// TIA Portal project "FactoryIO_Template_S7-1500_V15_V15.1" (V15.1)

(* hardware
DEVICE "S71500/ET200MP-Station_1"  S7-1500 station
   slot 0: "Profilschiene_0"  6ES7 590-1***0-0AA0
   slot 1: "PLC_1"  CPU 1511-1 PN  6ES7 511-1AK00-0AB0  V1.8
   slot 2: "AI 8xU/I/RTD/TC ST_1"  AI 8xU/I/RTD/TC ST  6ES7 531-7KF00-0AB0  V2.0
   slot 3: "AI 8xU/I/RTD/TC ST_2"  AI 8xU/I/RTD/TC ST  6ES7 531-7KF00-0AB0  V2.0
   slot 4: "AI 8xU/I/RTD/TC ST_3"  AI 8xU/I/RTD/TC ST  6ES7 531-7KF00-0AB0  V2.0
   slot 5: "AI 8xU/I/RTD/TC ST_4"  AI 8xU/I/RTD/TC ST  6ES7 531-7KF00-0AB0  V2.0
   slot 6: "DI 16x24VDC BA_1"  DI 16x24VDC BA  6ES7 521-1BH10-0AA0  V1.0
*)

// ===== PLC "PLC_1"  CPU 1511-1 PN =====

VAR_GLOBAL   // PLC tag table "Standard-Variablentabelle"
   "HighSensor" AT %E0.0 : Bool;
   "LowSensor" AT %I0.1 : Bool;
   "PalletSensor" AT %I0.2 : Bool;
   "Loaded" AT %I0.3 : Bool;
   "AtLeftEntry" AT %I0.4 : Bool;
   "AtLeftExit" AT %I0.5 : Bool;
   "AtRightEntry" AT %I0.6 : Bool;
   "AtRightExit" AT %I0.7 : Bool;
   "Start" AT %I1.0 : Bool;
   "Reset" AT %I1.1 : Bool;
   "Stop" AT %I1.2 : Bool;
   "EmergencyStop" AT %I1.3 : Bool;
   "Auto" AT %I1.4 : Bool;
   "Load" AT %Q0.1 : Bool;
   "Unload" AT %Q0.2 : Bool;
   "Transf. Left" AT %Q0.3 : Bool;
   "Transf. Right" AT %Q0.4 : Bool;
   "Conveyor Left" AT %Q0.5 : Bool;
   "Conveyor Right" AT %Q0.6 : Bool;
   "Start Light" AT %Q0.7 : Bool;
   "Reset Light" AT %Q1.0 : Bool;
   "Stop Light" AT %Q1.1 : Bool;
   "Counter" AT %QW30 : Int;
   "Conveyor Entry" AT %Q0.0 : Bool;
   "DelayReset" AT %T0 : Timer;
   "DelayTransferencia" AT %T1 : Timer;
END_VAR

TYPE "ControleDeCiclo"
   STRUCT
      Ciclo_Inicado : Bool;
      Em_Parada : Bool;
      Reset : Bool;
      Em_Manual : Bool;
      Em_Automatico : Bool;
      Counter_Entrada : Bool;
      Em_Anomali : Bool;
   END_STRUCT;
END_TYPE

// folder: SortByHeight

DATA_BLOCK "Painel_DB"   // DB1
{ S7_Optimized_Access := 'TRUE' }
VERSION : 0.1
// stored: InstanceOfName Painel
"Painel"
BEGIN
END_DATA_BLOCK

DATA_BLOCK "Conveyor_Entry_DB"   // DB2
{ S7_Optimized_Access := 'TRUE' }
VERSION : 0.1
// stored: InstanceOfName Conveyor_Entry
"Conveyor_Entry"
BEGIN
END_DATA_BLOCK

DATA_BLOCK "Controle_Sentido_DB"   // DB3
{ S7_Optimized_Access := 'TRUE' }
VERSION : 0.1
// stored: InstanceOfName Controle_Sentido
"Controle_Sentido"
BEGIN
END_DATA_BLOCK

// folder: (top level)

FUNCTION "MHJ-PLC-Lab-Function-S71500" : Void   // FC9000, SCL
{ S7_Optimized_Access := 'TRUE' }
VERSION : 0.1
   VAR_TEMP
      Value : Byte;
      ForCounter : Int;
   END_VAR
   VAR CONSTANT
      Value_01_DW : DWord := 16#1223_5486;
      Value_02_DW : DWord := 16#A6C9_D1F5;
   END_VAR
BEGIN

   #Value:=PEEK(area := 16#82,
        dbNumber := 0,
        byteOffset := 511);
   #Value := #Value + 1;

   POKE(area := 16#82,
        dbNumber := 0,
        byteOffset := 511,
        value := #Value);

   POKE(area := 16#82,
        dbNumber := 0,
        byteOffset := 1016,
        value := #Value_01_DW);
   POKE(area := 16#82,
        dbNumber := 0,
        byteOffset := 1020,
        value := #Value_02_DW);

   FOR #ForCounter := 0 TO 63 DO
       #Value:=PEEK(area := 16#1,
            dbNumber := 0,
            byteOffset := #ForCounter);
       POKE(area := 16#81,
            dbNumber := 0,
            byteOffset := #ForCounter,
            value := #Value);
   END_FOR;
   #Value := PEEK(area := 16#1,
                  dbNumber := 0,
                  byteOffset := 512);
   POKE(area := 16#82,
        dbNumber := 0,
        byteOffset := 512,
        value := #Value);
END_FUNCTION

ORGANIZATION_BLOCK "Main"   // OB1, FBD, ProgramCycle
TITLE = "Main Program Sweep (Cycle)"
{ S7_Optimized_Access := 'TRUE' }
VERSION : 0.1
   VAR_INPUT
      Initial_Call : Bool;   // Initial call of this OB
      Remanence : Bool;   // =True, if remanent data are available
   END_VAR
BEGIN

REGION Network 1
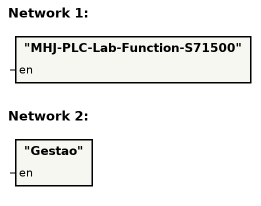
   "MHJ-PLC-Lab-Function-S71500"();
END_REGION

REGION Network 2
   "Gestao"();
END_REGION
END_ORGANIZATION_BLOCK

// folder: SortByHeight

FUNCTION "Gestao" : Void   // FC1, LAD
{ S7_Optimized_Access := 'TRUE' }
VERSION : 0.1
BEGIN

REGION Network 1
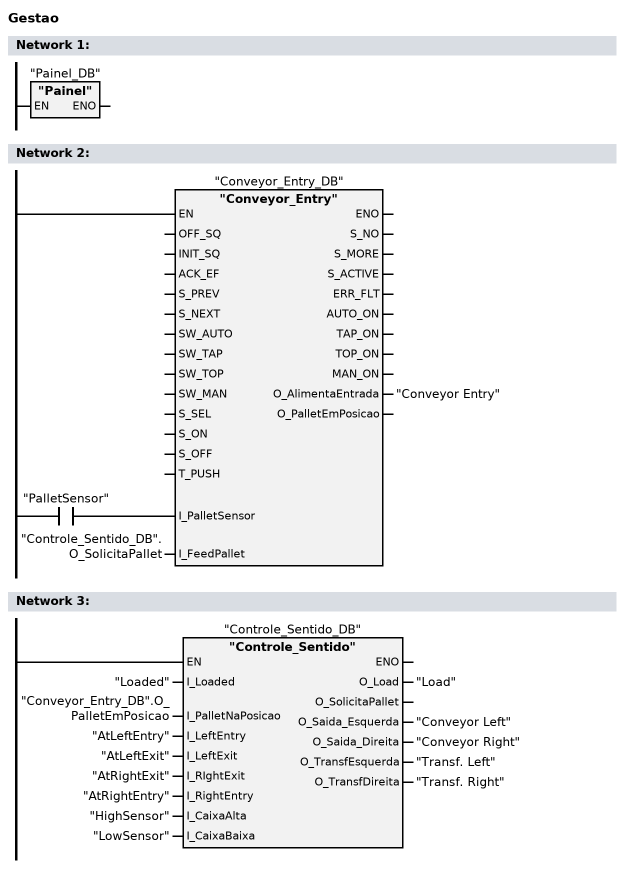
   RUNG wire#powerrail
      "Painel_DB"()
   END_RUNG
   // the same network as SCL:
   "Painel_DB"();   // "Painel"
END_REGION

REGION Network 2
   RUNG wire#powerrail
      "Conveyor_Entry_DB"(I_PalletSensor := wire#w1, OFF_SQ :=, INIT_SQ :=, ACK_EF :=, S_PREV :=, S_NEXT :=, SW_AUTO :=, SW_TAP :=, SW_TOP :=, SW_MAN :=, S_SEL :=, S_ON :=, S_OFF :=, T_PUSH :=, I_FeedPallet := "Controle_Sentido_DB".O_SolicitaPallet, S_NO =>, S_MORE =>, S_ACTIVE =>, ERR_FLT =>, AUTO_ON =>, TAP_ON =>, TOP_ON =>, MAN_ON =>, O_AlimentaEntrada => "Conveyor Entry", O_PalletEmPosicao =>)
   END_RUNG
   RUNG wire#powerrail
      Contact( "PalletSensor" )
   END_RUNG wire#w1
   // the same network as SCL:
   "Conveyor_Entry_DB"(I_PalletSensor := "PalletSensor",   // "Conveyor_Entry"
                       I_FeedPallet := "Controle_Sentido_DB".O_SolicitaPallet,
                       O_AlimentaEntrada => "Conveyor Entry");
END_REGION

REGION Network 3
   RUNG wire#powerrail
      "Controle_Sentido_DB"(I_Loaded := "Loaded", I_PalletNaPosicao := "Conveyor_Entry_DB".O_PalletEmPosicao, I_LeftEntry := "AtLeftEntry", I_LeftExit := "AtLeftExit", I_RIghtExit := "AtRightExit", I_RightEntry := "AtRightEntry", I_CaixaAlta := "HighSensor", I_CaixaBaixa := "LowSensor", O_Load => "Load", O_SolicitaPallet =>, O_Saida_Esquerda => "Conveyor Left", O_Saida_Direita => "Conveyor Right", O_TransfEsquerda => "Transf. Left", O_TransfDireita => "Transf. Right")
   END_RUNG
   // the same network as SCL:
   "Controle_Sentido_DB"(I_Loaded := "Loaded",   // "Controle_Sentido"
                         I_PalletNaPosicao := "Conveyor_Entry_DB".O_PalletEmPosicao,
                         I_LeftEntry := "AtLeftEntry",
                         I_LeftExit := "AtLeftExit",
                         I_RIghtExit := "AtRightExit",
                         I_RightEntry := "AtRightEntry",
                         I_CaixaAlta := "HighSensor",
                         I_CaixaBaixa := "LowSensor",
                         O_Load => "Load",
                         O_Saida_Esquerda => "Conveyor Left",
                         O_Saida_Direita => "Conveyor Right",
                         O_TransfEsquerda => "Transf. Left",
                         O_TransfDireita => "Transf. Right");
END_REGION
END_FUNCTION

// folder: SortByHeight/ControleSentido

FUNCTION_BLOCK "Controle_Sentido"   // FB3, LAD
{ S7_Optimized_Access := 'TRUE' }
VERSION : 0.1
   VAR_INPUT
      I_Loaded : Bool;
      I_PalletNaPosicao : Bool;
      I_LeftEntry : Bool;
      I_LeftExit : Bool;
      I_RIghtExit : Bool;
      I_RightEntry : Bool;
      I_CaixaAlta : Bool;
      I_CaixaBaixa : Bool;
   END_VAR
   VAR_OUTPUT
      O_Load : Bool;
      O_SolicitaPallet : Bool;
      O_Saida_Esquerda : Bool;
      O_Saida_Direita : Bool;
      O_TransfEsquerda : Bool;
      O_TransfDireita : Bool;
   END_VAR
   VAR
      Abastecido : Bool;
      Desabastecido : Bool;
      Estado_Saida_Esquerda : Bool;
      Estado_Saida_Direita : Bool;
      "Caixa alta" : Bool;
      "Caixa baixa" : Bool;
      M1 : Bool;
      M2 : Bool;
      M3 : Bool;
      M4 : Bool;
      M5 : Bool;
      M6 : Bool;
      Transf_Esquerda : Bool;
      Transf_Direita : Bool;
      Em_Transferencia : Bool;
      StoptEsquerda : Bool;
      StoptDireita : Bool;
   END_VAR
   VAR_TEMP   // added for the SCL form of the ladder/FBD networks
      _w1 : Bool;
   END_VAR
BEGIN

REGION Network 1: ############## ABASTECIMENTO ################
END_REGION

REGION Network 2: Desabastecido
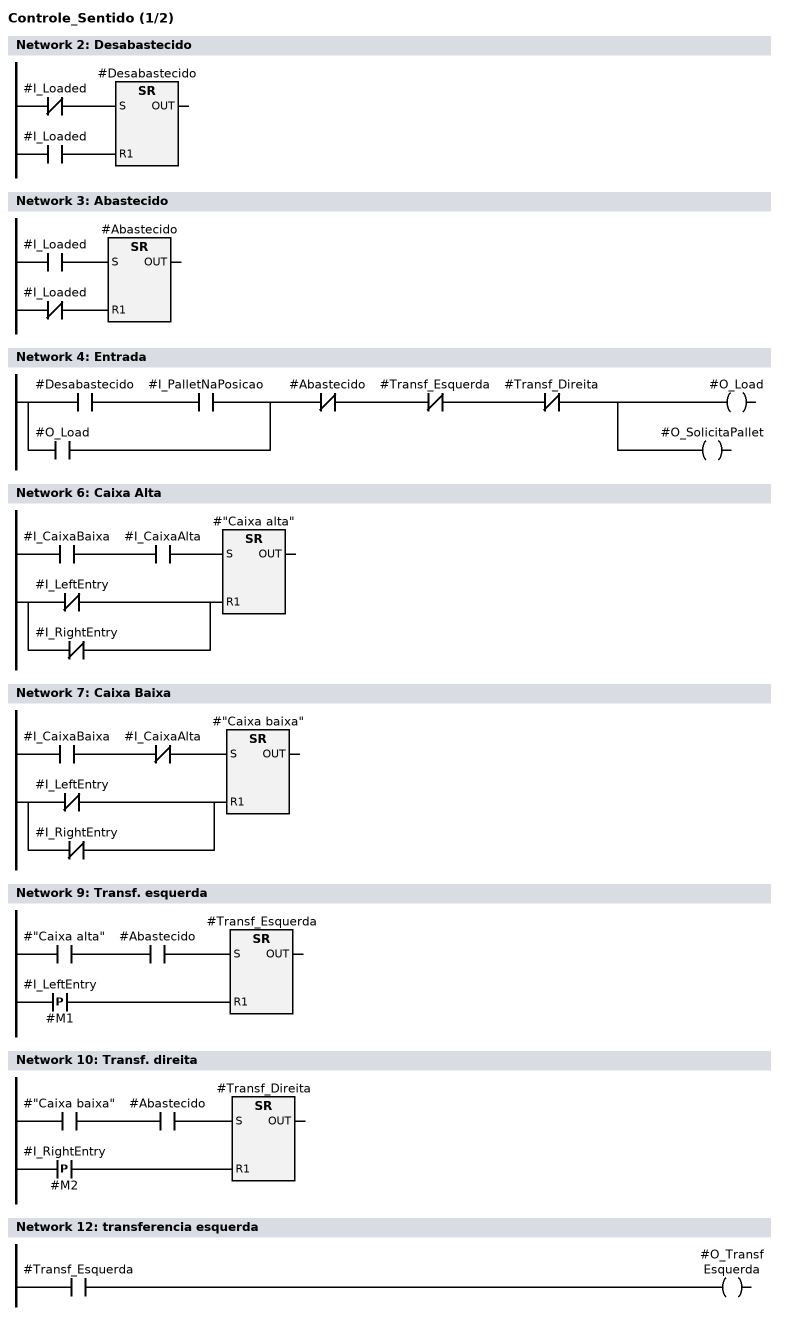
   RUNG wire#powerrail
      I_Contact( #I_Loaded )
      S_SR(operand := #Desabastecido, r1 := wire#w1)
   END_RUNG
   RUNG wire#powerrail
      Contact( #I_Loaded )
   END_RUNG wire#w1
   // the same network as SCL:
   IF NOT #I_Loaded THEN
       #Desabastecido := TRUE;   // SR flip-flop
   END_IF;
   IF #I_Loaded THEN #Desabastecido := FALSE; END_IF;
END_REGION

REGION Network 3: Abastecido
   RUNG wire#powerrail
      Contact( #I_Loaded )
      S_SR(operand := #Abastecido, r1 := wire#w1)
   END_RUNG
   RUNG wire#powerrail
      I_Contact( #I_Loaded )
   END_RUNG wire#w1
   // the same network as SCL:
   IF #I_Loaded THEN
       #Abastecido := TRUE;   // SR flip-flop
   END_IF;
   IF NOT #I_Loaded THEN #Abastecido := FALSE; END_IF;
END_REGION

REGION Network 4: Entrada
   RUNG wire#powerrail
      Contact( #Desabastecido )
      Contact( #I_PalletNaPosicao )
      wire#w1
      I_Contact( #Abastecido )
      I_Contact( #Transf_Esquerda )
      I_Contact( #Transf_Direita )
      wire#w2
      Coil( #O_Load )
   END_RUNG
   RUNG wire#powerrail
      Contact( #O_Load )
   END_RUNG wire#w1
   RUNG wire#w2
      Coil( #O_SolicitaPallet )
   END_RUNG
   // the same network as SCL:
   #O_Load := ((#Desabastecido AND #I_PalletNaPosicao) OR #O_Load) AND NOT #Abastecido AND NOT #Transf_Esquerda AND NOT #Transf_Direita;
   #O_SolicitaPallet := #O_Load;
END_REGION

REGION Network 5: ################ TAMANHOS #################
END_REGION

REGION Network 6: Caixa Alta
   RUNG wire#powerrail
      Contact( #I_CaixaBaixa )
      Contact( #I_CaixaAlta )
      S_SR(operand := #"Caixa alta", r1 := wire#w1)
   END_RUNG
   RUNG wire#powerrail
      I_Contact( #I_LeftEntry )
   END_RUNG wire#w1
   RUNG wire#powerrail
      I_Contact( #I_RightEntry )
   END_RUNG wire#w1
   // the same network as SCL:
   IF #I_CaixaBaixa AND #I_CaixaAlta THEN
       #"Caixa alta" := TRUE;   // SR flip-flop
   END_IF;
   IF NOT #I_LeftEntry OR NOT #I_RightEntry THEN #"Caixa alta" := FALSE; END_IF;
END_REGION

REGION Network 7: Caixa Baixa
   RUNG wire#powerrail
      Contact( #I_CaixaBaixa )
      I_Contact( #I_CaixaAlta )
      S_SR(operand := #"Caixa baixa", r1 := wire#w1)
   END_RUNG
   RUNG wire#powerrail
      I_Contact( #I_LeftEntry )
   END_RUNG wire#w1
   RUNG wire#powerrail
      I_Contact( #I_RightEntry )
   END_RUNG wire#w1
   // the same network as SCL:
   IF #I_CaixaBaixa AND NOT #I_CaixaAlta THEN
       #"Caixa baixa" := TRUE;   // SR flip-flop
   END_IF;
   IF NOT #I_LeftEntry OR NOT #I_RightEntry THEN #"Caixa baixa" := FALSE; END_IF;
END_REGION

REGION Network 8: ############## TRANFERENCIAS ################
END_REGION

REGION Network 9: Transf. esquerda
   RUNG wire#powerrail
      Contact( #"Caixa alta" )
      Contact( #Abastecido )
      S_SR(operand := #Transf_Esquerda, r1 := wire#w1)
   END_RUNG
   RUNG wire#powerrail
      P_Contact(operand := #I_LeftEntry, bit := #M1)
   END_RUNG wire#w1
   // the same network as SCL:
   #_w1 := #I_LeftEntry AND NOT #M1;   // rising edge of #I_LeftEntry
   #M1 := #I_LeftEntry;
   IF #"Caixa alta" AND #Abastecido THEN
       #Transf_Esquerda := TRUE;   // SR flip-flop
   END_IF;
   IF #_w1 THEN #Transf_Esquerda := FALSE; END_IF;
END_REGION

REGION Network 10: Transf. direita
   RUNG wire#powerrail
      Contact( #"Caixa baixa" )
      Contact( #Abastecido )
      S_SR(operand := #Transf_Direita, r1 := wire#w1)
   END_RUNG
   RUNG wire#powerrail
      P_Contact(operand := #I_RightEntry, bit := #M2)
   END_RUNG wire#w1
   // the same network as SCL:
   #_w1 := #I_RightEntry AND NOT #M2;   // rising edge of #I_RightEntry
   #M2 := #I_RightEntry;
   IF #"Caixa baixa" AND #Abastecido THEN
       #Transf_Direita := TRUE;   // SR flip-flop
   END_IF;
   IF #_w1 THEN #Transf_Direita := FALSE; END_IF;
END_REGION

REGION Network 11: ################# SAIDA ###################
END_REGION

REGION Network 12: transferencia esquerda
   RUNG wire#powerrail
      Contact( #Transf_Esquerda )
      Coil( #O_TransfEsquerda )
   END_RUNG
   // the same network as SCL:
   #O_TransfEsquerda := #Transf_Esquerda;
END_REGION

REGION Network 13: Conveyor esquerda
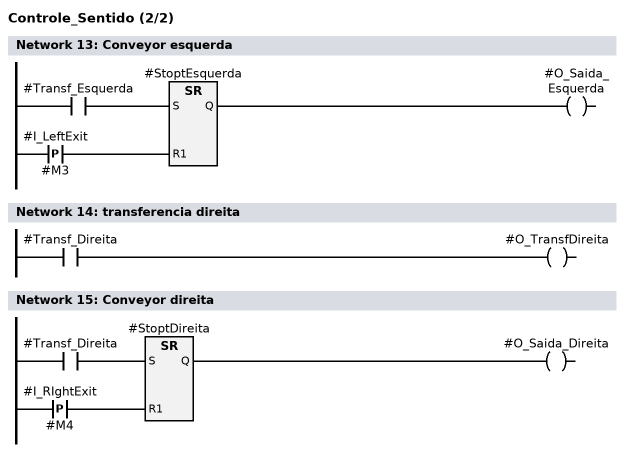
   RUNG wire#powerrail
      Contact( #Transf_Esquerda )
      S_SR(operand := #StoptEsquerda, r1 := wire#w1)
      Coil( #O_Saida_Esquerda )
   END_RUNG
   RUNG wire#powerrail
      P_Contact(operand := #I_LeftExit, bit := #M3)
   END_RUNG wire#w1
   // the same network as SCL:
   #_w1 := #I_LeftExit AND NOT #M3;   // rising edge of #I_LeftExit
   #M3 := #I_LeftExit;
   IF #Transf_Esquerda THEN
       #StoptEsquerda := TRUE;   // SR flip-flop
   END_IF;
   IF #_w1 THEN #StoptEsquerda := FALSE; END_IF;
   #O_Saida_Esquerda := #StoptEsquerda;
END_REGION

REGION Network 14: transferencia direita
   RUNG wire#powerrail
      Contact( #Transf_Direita )
      Coil( #O_TransfDireita )
   END_RUNG
   // the same network as SCL:
   #O_TransfDireita := #Transf_Direita;
END_REGION

REGION Network 15: Conveyor direita
   RUNG wire#powerrail
      Contact( #Transf_Direita )
      S_SR(operand := #StoptDireita, r1 := wire#w1)
      Coil( #O_Saida_Direita )
   END_RUNG
   RUNG wire#powerrail
      P_Contact(operand := #I_RIghtExit, bit := #M4)
   END_RUNG wire#w1
   // the same network as SCL:
   #_w1 := #I_RIghtExit AND NOT #M4;   // rising edge of #I_RIghtExit
   #M4 := #I_RIghtExit;
   IF #Transf_Direita THEN
       #StoptDireita := TRUE;   // SR flip-flop
   END_IF;
   IF #_w1 THEN #StoptDireita := FALSE; END_IF;
   #O_Saida_Direita := #StoptDireita;
END_REGION
END_FUNCTION_BLOCK

// folder: SortByHeight/ConveyorEntry

FUNCTION_BLOCK "Conveyor_Entry"   // FB2, GRAPH_PLUS
{ S7_Optimized_Access := 'TRUE' }
VERSION : 0.1
   VAR_INPUT
      OFF_SQ : Bool := false;   // Turn sequence off
      INIT_SQ : Bool := false;   // Set sequence to initial state
      ACK_EF : Bool := false;   // Acknowledge all errors and faults
      S_PREV : Bool := false;   // Output previous step in parameter S_NO
      S_NEXT : Bool := false;   // Indicate next step in parameter S_NO
      SW_AUTO : Bool := false;   // Automatic mode
      SW_TAP : Bool := false;   // Semiautomatic/switch with transition
      SW_TOP : Bool := false;   // Semiautomatic/ignore transition
      SW_MAN : Bool := false;   // Manual mode
      S_SEL : Int := 0;   // Select step to be output to S_NO
      S_ON : Bool := false;   // Activate step indicated in S_NO
      S_OFF : Bool := false;   // Deactivate step indicated S_NO
      T_PUSH : Bool := false;   // Enable transition to switch in semi automatic mode
      I_PalletSensor : Bool;
      I_FeedPallet : Bool;
   END_VAR
   VAR_OUTPUT
      S_NO : Int := 0;   // Step number
      S_MORE : Bool := false;   // More steps are available and can be shown in S_NO
      S_ACTIVE : Bool := false;   // Step indicated in S_NO is active
      ERR_FLT : Bool := false;   // Interlock or supervision group error
      AUTO_ON : Bool := false;   // Automatic mode is active
      TAP_ON : Bool := false;   // Semiautomatic mode/step with transition enabled
      TOP_ON : Bool := false;   // Semiautomatic mode/ignore transition enabled
      MAN_ON : Bool := false;   // Manual mode is active
      O_AlimentaEntrada : Bool;
      O_PalletEmPosicao : Bool;
   END_VAR
   VAR
      HMI_INFO : Array[0..8] of UInt;
      IF_PAR : G7_IfParPlus_V2;
      RT_DATA : G7_RTDataPlus_V2;   // Internal data area
      Trans4 : G7_TransitionPlus_V2;   // Transition structure
      Trans1 : G7_TransitionPlus_V2;   // Transition structure
      Trans2 : G7_TransitionPlus_V2;   // Transition structure
      Trans3 : G7_TransitionPlus_V2;   // Transition structure
      Step4 : G7_StepPlus_V2;   // Step structure
      Step1 : G7_StepPlus_V2;   // Step structure
      Step2 : G7_StepPlus_V2;   // Step structure
      Step3 : G7_StepPlus_V2;   // Step structure
      SINI : Array[0..1] of USInt;
      LSTT : Array[0..3] of USInt;
      ATAJ : Array[0..3] of USInt;
      ATAB : Array[0..3] of USInt;
      PSTT : Array[0..3] of USInt;
      NSTT : Array[0..3] of USInt;
      ASSJ : Array[0..3] of USInt;
      ASSB : Array[0..3] of USInt;
      PTTS : Array[0..3] of USInt;
      NTTS : Array[0..3] of USInt;
      SW_SQTS : Array[0..3] of USInt;
      SWITCH : Array[0..0] of USInt;
      TVX : Array[0..1] of USInt;
      TTX : Array[0..1] of USInt;
      TSX : Array[0..1] of USInt;
      S00X : Array[0..1] of USInt;
      SOFFX : Array[0..1] of USInt;
      SONX : Array[0..1] of USInt;
      SAX : Array[0..1] of USInt;
      SERRX : Array[0..4] of USInt;
      SMX : Array[0..4] of USInt;
      S0X : Array[0..4] of USInt;
      S1X : Array[0..4] of USInt;
      IL_ALARM_INST : Program_Alarm;
      SUP_ALARM_INST : Program_Alarm;
      STEP_TIME_ALARM_INST : Program_Alarm;
      IEC_TIMER_INST : IEC_TIMER;
      TRANSACTION_FLAG : Bool := false;
   END_VAR
   // LSTT[3] := 1;
   // SINI[0] := 2;
   // LSTT[0] := 255;
   // LSTT[1] := 255;
   // ATAJ[3] := 3;
   // ATAJ[1] := 1;
   // ATAJ[2] := 2;
   // ATAB[3] := 3;
   // ATAB[1] := 1;
   // ATAB[2] := 2;
   // PSTT[3] := 3;
   // PSTT[1] := 1;
   // PSTT[2] := 2;
   // ASSJ[3] := 3;
   // NSTT[0] := 1;
   // NSTT[1] := 2;
   // LSTT[2] := 255;
   // ASSJ[1] := 1;
   // ASSJ[2] := 2;
   // ASSB[3] := 3;
   // ASSB[1] := 1;
   // ASSB[2] := 2;
   // SINI[1] := 1;
   // PTTS[0] := 255;
   // PTTS[2] := 1;
   // NTTS[3] := 3;
   // NTTS[1] := 1;
   // NTTS[2] := 2;
   // PTTS[3] := 2;
   // TVX[0] := 16#1;
   // TTX[0] := 16#1;
   // TSX[0] := 16#1;
   // S00X[0] := 16#1;
   // SOFFX[0] := 16#1;
   // SONX[0] := 16#1;
   // SAX[0] := 16#1;
   // SERRX[0] := 16#1;
   // SMX[0] := 16#1;
   // S0X[0] := 16#1;
   // S1X[0] := 16#1;
   // NSTT[2] := 3;
   // NSTT[3] := 1;
BEGIN
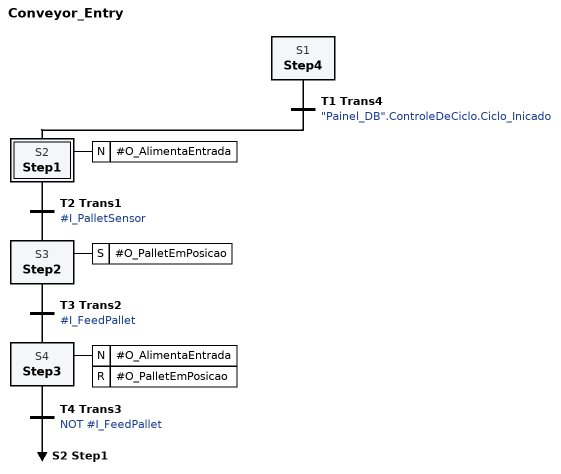
   // sequencer 1
   INITIAL_STEP Step1:   // S2, max time T#10S, warning time T#7S
              N    #O_AlimentaEntrada
   END_STEP
   TRANSITION Trans1 FROM Step1 TO Step2   // T2
      := #I_PalletSensor;
   END_TRANSITION
   STEP Step2:   // S3, max time T#10S, warning time T#7S
              S    #O_PalletEmPosicao
   END_STEP
   TRANSITION Trans2 FROM Step2 TO Step3   // T3
      := #I_FeedPallet;
   END_TRANSITION
   STEP Step3:   // S4, max time T#10S, warning time T#7S
              N    #O_AlimentaEntrada
              R    #O_PalletEmPosicao
   END_STEP
   TRANSITION Trans3 FROM Step3 TO Step1   // T4, jump
      := NOT #I_FeedPallet;
   END_TRANSITION
   STEP Step4:   // S1, max time T#10S, warning time T#7S
   END_STEP
   TRANSITION Trans4 FROM Step4 TO Step1   // T1
      := "Painel_DB".ControleDeCiclo.Ciclo_Inicado;
   END_TRANSITION
END_FUNCTION_BLOCK

// folder: SortByHeight/Painel

FUNCTION_BLOCK "Painel"   // FB1, LAD
{ S7_Optimized_Access := 'TRUE' }
VERSION : 0.1
   VAR
      ControleDeCiclo : "ControleDeCiclo";
   END_VAR
BEGIN

REGION Network 1: Btn start
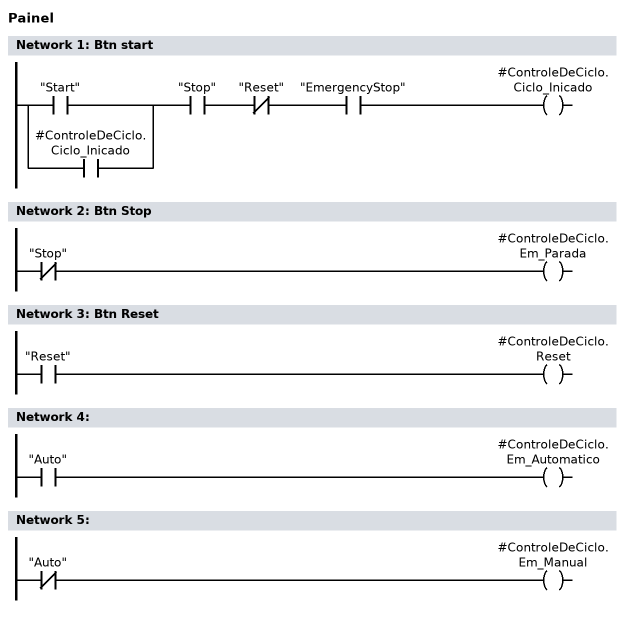
   RUNG wire#powerrail
      Contact( "Start" )
      wire#w1
      Contact( "Stop" )
      I_Contact( "Reset" )
      Contact( "EmergencyStop" )
      Coil( #ControleDeCiclo.Ciclo_Inicado )
   END_RUNG
   RUNG wire#powerrail
      Contact( #ControleDeCiclo.Ciclo_Inicado )
   END_RUNG wire#w1
   // the same network as SCL:
   #ControleDeCiclo.Ciclo_Inicado := ("Start" OR #ControleDeCiclo.Ciclo_Inicado) AND "Stop" AND NOT "Reset" AND "EmergencyStop";
END_REGION

REGION Network 2: Btn Stop
   RUNG wire#powerrail
      I_Contact( "Stop" )
      Coil( #ControleDeCiclo.Em_Parada )
   END_RUNG
   // the same network as SCL:
   #ControleDeCiclo.Em_Parada := NOT "Stop";
END_REGION

REGION Network 3: Btn Reset
   RUNG wire#powerrail
      Contact( "Reset" )
      Coil( #ControleDeCiclo.Reset )
   END_RUNG
   // the same network as SCL:
   #ControleDeCiclo.Reset := "Reset";
END_REGION

REGION Network 4
   RUNG wire#powerrail
      Contact( "Auto" )
      Coil( #ControleDeCiclo.Em_Automatico )
   END_RUNG
   // the same network as SCL:
   #ControleDeCiclo.Em_Automatico := "Auto";
END_REGION

REGION Network 5
   RUNG wire#powerrail
      I_Contact( "Auto" )
      Coil( #ControleDeCiclo.Em_Manual )
   END_RUNG
   // the same network as SCL:
   #ControleDeCiclo.Em_Manual := NOT "Auto";
END_REGION
END_FUNCTION_BLOCK